FUNCTION_BLOCK FB_BandZonderKlep
VAR_INPUT
	i_eState 		: eSingleState;
	i_xGoHold 		: BOOL; //keep pallet on band
	i_xGoEmpty		: BOOL; //move pallet to other segment
	i_xAlarmReset	: BOOL;
END_VAR
VAR_OUTPUT
	o_xMotor 		: BOOL := FALSE;
	o_xErrorMotor 	: BOOL := FALSE;
	o_xAlarmMotor 	: BOOL := FALSE;
	o_xGivingToNext	: BOOL;
END_VAR
VAR
END_VAR

// Van Emma

END_FUNCTION_BLOCK

(* stored: Version 1.1.0.1
   POU FB_BandZonderKlep: Id {6f0d6422-6ccd-4d17-bba5-56fca414051a}, SpecialFunc None *)
